// TIA Portal V21 export
DATA_BLOCK "Axis_1"   // DB3
VERSION : 1.0
// stored: InstanceOfName AxisAS_Mng_v2.0, InstanceOfType FB
"AxisAS_Mng_v2.0"
   // VAR RETAIN
   //    DataIn : "AxixAS_DataIn_Type_v2.0";
   //    DataOut : "AxixAS_DataOut_Type_v2.0";
   // END_VAR
   // VAR
   //    Sincro { S7_SetPoint := 'True'} : "AxixAS_DataSincro_Type_v2.0";
   // END_VAR
   // VAR RETAIN
   //    Cfg { S7_SetPoint := 'True'} : "AxixAS_CFG_Type_v2.0";   // Configurazione Asse
   //    Work : Struct   // Gestione interna Asse
   //       xEnablePos { S7_SetPoint := 'True'} : Bool := FALSE;
   //       xINEnable : Bool := FALSE;
   //       xDriveReady { S7_SetPoint := 'True'} : Bool := FALSE;
   //       xCmdVirSpeedChanged { S7_SetPoint := 'True'} : Bool := FALSE;
   //       "xCurveS-L" { ExternalWritable := 'False'; S7_SetPoint := 'True'} : Bool := TRUE;
   //       "xAutoChangeS-L" { S7_SetPoint := 'True'} : Bool := FALSE;
   //       "xCTRAutoChangeS-L" { S7_SetPoint := 'True'} : Bool := FALSE;
   //       xDecStop { S7_SetPoint := 'True'} : Bool := FALSE;
   //       xDecResearch { S7_SetPoint := 'True'} : Bool := FALSE;
   //       xStopVirPositioner { S7_SetPoint := 'True'} : Bool := TRUE;
   //       xEnableJog { S7_SetPoint := 'True'} : Bool := FALSE;
   //       xChangeTargetPulse { S7_SetPoint := 'True'} : Bool := FALSE;
   //       xAutoSpeedPulse { S7_SetPoint := 'True'} : Bool := FALSE;
   //       xEnablePulse { S7_SetPoint := 'True'} : Bool := FALSE;
   //       f_PositionTarget { S7_SetPoint := 'True'} : Real := 2222.0;
   //       fVirPos { S7_SetPoint := 'True'} : Real := 2221.003;
   //       f_SpeedReqCalc { S7_SetPoint := 'True'} : Real := 500.0;
   //       fVirSpeed { S7_SetPoint := 'True'} : Real := 0.0;
   //       fVirSpeedLinear { S7_SetPoint := 'True'} : Real := 0.0;
   //       fVirSpeedLog { S7_SetPoint := 'True'} : Real := 0.0;
   //       fVirSpeedCos { S7_SetPoint := 'True'} : Real := 0.0;
   //       fCmdVirSpeed { S7_SetPoint := 'True'} : Real := 0.0;
   //       fCmdVirSpeedMemo { S7_SetPoint := 'True'} : Real := 0.0;
   //       fCmdVirAcc { S7_SetPoint := 'True'} : Real := 5.068141;
   //       fCmdVirDec { S7_SetPoint := 'True'} : Real := 4.054513;
   //       fLimVirDec { S7_SetPoint := 'True'} : Real := 0.0;
   //       fDecVirStop { S7_SetPoint := 'True'} : Real := 0.0;
   //       fCalcEncErr { S7_SetPoint := 'True'} : Real := 0.0;
   //       fJogSpeed { S7_SetPoint := 'True'} : Real := 0.0;
   //       fCmdJogSpeed { S7_SetPoint := 'True'} : Real := 0.0;
   //       fCmdJogAcc { S7_SetPoint := 'True'} : Real := 0.0;
   //       fCmdJogDec { S7_SetPoint := 'True'} : Real := 0.0;
   //       "fLim+Ppid" { S7_SetPoint := 'True'} : Real := 240.0;
   //       "fLim-Ppid" { S7_SetPoint := 'True'} : Real := -240.0;
   //       fOutSpeedMot { S7_SetPoint := 'True'} : Real := 0.0;
   //       fSuppCalcPpid { S7_SetPoint := 'True'} : Real := 5.0;
   //       fMemoMaxSpeed { S7_SetPoint := 'True'} : Real := 1.0;
   //       fPpid { S7_SetPoint := 'True'} : Real := 0.0;
   //       fMemoOldPos { S7_SetPoint := 'True'} : Real := 2222.0;
   //       fAccOnWork { S7_SetPoint := 'True'} : Real := 1000.0;
   //       fDecOnWork { S7_SetPoint := 'True'} : Real := 800.0;
   //       fSpaceFromTarget : Real := 0.0;
   //       xTimBrakeDelay_Fwd : Bool := FALSE;
   //       xTimBrakeDelay_Bkw : Bool := FALSE;
   //       xTimStopEndPos : Bool := FALSE;
   //       xMotorMagn_pulse : Bool := FALSE;
   //       fCalc : Array[0..20] of Real;
   //       xCalc : Array[0..20] of Bool;
   //    END_STRUCT;
   // END_VAR
   // VAR
   //    TmrBrake_Fwd : IEC_TIMER;   // Timer sgancio freno FWD
   //    TmrBrake_Bkw : IEC_TIMER;   // Timer sgancio freno BKW
   //    Tmr_EndPos : IEC_TIMER;   // Timer allarme controllo fine posizionamento
   //    Tmr_DriveOnReq : IEC_TIMER;   // Timer OFF richiesta Drive Ready
   //    Tmr_DriveOffReq : IEC_TIMER;
   //    Tmr_OnMove : IEC_TIMER;
   // END_VAR
BEGIN
   DataIn.ixEnablePos := FALSE;
   DataIn.ixDriveReady := FALSE;
   DataIn.ixEnableLevRes := FALSE;
   DataIn.ixLevelReached := FALSE;
   DataIn.ixMotorReadyReq := FALSE;
   DataIn.ixAlarmReset := FALSE;
   DataIn.ixAbort := FALSE;
   DataIn.ixJogPos := FALSE;
   DataIn.ixJogNeg := FALSE;
   DataIn.xAutoSpeedDetect := FALSE;
   DataIn.xAutoAccDecCalculation := FALSE;
   DataIn.ifPositionRequest := 2222.0;
   DataIn.ifSpeedRequest := 500.0;
   DataIn.ifPositionStartLev := 500.0;
   DataIn.ifSpeedLev := 100.0;
   DataIn.ifAccRamp := 1000.0;
   DataIn.ifDecRamp := 1000.0;
   DataIn.ifTimeScan := 0.005068141;
   DataIn.ifEncoder := 2221.003;
   DataOut.oxCmdMotorForw := FALSE;
   DataOut.oxCmdMotorBack := FALSE;
   DataOut.oxCmdBrake := FALSE;
   DataOut.oxPosError := FALSE;
   DataOut.oxSincroError := FALSE;
   DataOut.oxEndPos := TRUE;
   DataOut.oxEndPosBig := TRUE;
   DataOut.oxStopSpeed := TRUE;
   DataOut.oxAccOnWork := FALSE;
   DataOut.oxDecOnWork := FALSE;
   DataOut.ofSpeedRequest := 0.0;
   DataOut.ofEncMotorPos := 2221.003;
   DataOut.ofMaxError := 0.0;
   DataOut.ofSpaceStop := 2.0;
   DataOut.ofSpaceLevRes := 43.75;
   DataOut.ofSpaceStart := 125.0;
   DataOut.otTimeMove := T#8S_555MS;
   Sincro.DataIn.ixEnablePos := FALSE;
   Sincro.DataIn.ixDriveReady := FALSE;
   Sincro.DataIn.ixEnableLevRes := FALSE;
   Sincro.DataIn.ixLevelReached := FALSE;
   Sincro.DataIn.ixMotorReadyReq := FALSE;
   Sincro.DataIn.ixAlarmReset := FALSE;
   Sincro.DataIn.ixAbort := FALSE;
   Sincro.DataIn.ixJogPos := FALSE;
   Sincro.DataIn.ixJogNeg := FALSE;
   Sincro.DataIn.xAutoSpeedDetect := FALSE;
   Sincro.DataIn.xAutoAccDecCalculation := FALSE;
   Sincro.DataIn.ifPositionRequest := 0.0;
   Sincro.DataIn.ifSpeedRequest := 0.0;
   Sincro.DataIn.ifPositionStartLev := 0.0;
   Sincro.DataIn.ifSpeedLev := 0.0;
   Sincro.DataIn.ifAccRamp := 0.0;
   Sincro.DataIn.ifDecRamp := 0.0;
   Sincro.DataIn.ifTimeScan := 0.0;
   Sincro.DataIn.ifEncoder := 0.0;
   Sincro.DataOut.oxCmdMotorForw := FALSE;
   Sincro.DataOut.oxCmdMotorBack := FALSE;
   Sincro.DataOut.oxCmdBrake := FALSE;
   Sincro.DataOut.oxPosError := FALSE;
   Sincro.DataOut.oxSincroError := FALSE;
   Sincro.DataOut.oxEndPos := FALSE;
   Sincro.DataOut.oxEndPosBig := FALSE;
   Sincro.DataOut.oxStopSpeed := FALSE;
   Sincro.DataOut.oxAccOnWork := FALSE;
   Sincro.DataOut.oxDecOnWork := FALSE;
   Sincro.DataOut.ofSpeedRequest := 0.0;
   Sincro.DataOut.ofEncMotorPos := 0.0;
   Sincro.DataOut.ofMaxError := 0.0;
   Sincro.DataOut.ofSpaceStop := 0.0;
   Sincro.DataOut.ofSpaceLevRes := 0.0;
   Sincro.DataOut.ofSpaceStart := 0.0;
   Sincro.DataOut.otTimeMove := T#0MS;
   Sincro.ixEnableSincro := 0;
   Sincro."ifDistance_Master/Slave" := 0.0;
   Sincro.ifErrorSincro := 0.0;
   Cfg.fJogSpeed := 10.0;
   Cfg.fJogAcc := 10.0;
   Cfg.fJogDec := 10.0;
   Cfg.fVirt_EncWindPos := 1.0;
   Cfg.fMotWindPos := 2.0;
   Cfg.fMotWindPosBig := 30.0;
   Cfg.fMaxErrEnc := 10.0;
   Cfg.fMaxSpeed := 1200.0;
   Cfg.fMinAccRamp := 100.0;
   Cfg.fMinDecRamp := 100.0;
   Cfg.fMaxAccRamp := 1200.0;
   Cfg.fMaxDecRamp := 800.0;
   Cfg.fThreshold_SUP_AutoSpeed := 500.0;
   Cfg.fThreshold_INF_AutoSpeed := 0.0;
   Cfg."xCurveS-L" := 2;
   Cfg.fMotWindSpeed := 10.0;
   Cfg.fMotAdvStopPosition := 0.0;
   Cfg.fKPpid_Pos := 1.0;
   Cfg.fKPpidAcc_Pos := 1.0;
   Cfg.fKPpidDec_Pos := 4.0;
   Cfg.fKPpid_Vel := 1.0;
   Cfg.fKPpidAcc_Vel := 1.0;
   Cfg.fKPpidDec_Vel := 1.0;
   Cfg.fMinSpeed := 20.0;
   Cfg.fFirstStepNepero := 6.0;
   Cfg."fAutoChangeS-Lvalue" := 0.0;
   Cfg.tBrakeDelay_Fwd := T#100MS;
   Cfg.tBrakeDelay_Bkw := T#100MS;
   Cfg.tDriveOnReq := T#5S;
   Cfg.tCtrEndPos := T#1S;
   Cfg.xDisablePos := FALSE;
   Work.fCalc[0..19] := 0.0;
   Work.fCalc[20] := 1617.987;
   Work.xCalc[0] := TRUE;
   Work.xCalc[1..20] := FALSE;
   TmrBrake_Fwd.PT := T#100MS;
   TmrBrake_Fwd.IN := FALSE;
   TmrBrake_Bkw.PT := T#100MS;
   TmrBrake_Bkw.IN := FALSE;
   Tmr_EndPos.PT := T#1S;
   Tmr_EndPos.IN := FALSE;
   Tmr_DriveOnReq.PT := T#5S;
   Tmr_DriveOnReq.IN := FALSE;
   Tmr_DriveOffReq.PT := T#5S;
   Tmr_DriveOffReq.IN := FALSE;
   Tmr_OnMove.PT := T#1M_40S;
   Tmr_OnMove.IN := FALSE;
END_DATA_BLOCK
